ABB RAPID module: Module1.mod

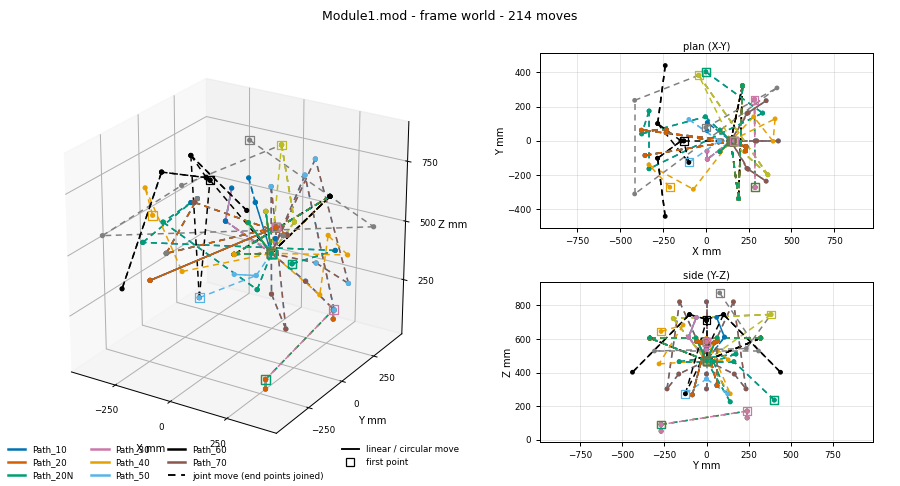
[picture p0: tool path of Module1.mod in frame world, 214 of 214 moves have a stored position in this frame; points joined in program order, loops and branches not executed]
MODULE Module1
    CONST robtarget p1:=[[392.068313627,0,352.752670777],[0,-0.707106781,0.707106781,0],[0,0,-1,0],[90,9E+09,9E+09,9E+09,9E+09,9E+09]];
    CONST robtarget p2:=[[0.889574022,-392.067304437,352.752670777],[0,-0.001134464,0.999999356,0],[-1,0,-1,0],[0.629463871,9E+09,9E+09,9E+09,9E+09,9E+09]];
    CONST robtarget p3:=[[218.23553446,-1.336915589,746.107847434],[0.698810372,0.082286187,0.062863115,0.707772051],[0,2,-1,4],[90.000000666,9E+09,9E+09,9E+09,9E+09,9E+09]];
    CONST robtarget Target_10:=[[521.001806146,0.000051805,471.113280829],[0.087155634,0.000000007,-0.996194708,0.000000054],[-2,1,0,4],[36.59813987,9E+09,9E+09,9E+09,9E+09,9E+09]];
    CONST robtarget Target_20:=[[285.146257362,-272.870516499,35.963966592],[0.000757376,0.999985094,-0.005407215,0.000030026],[-2,1,1,4],[5.849592085,9E+09,9E+09,9E+09,9E+09,9E+09]];
    CONST robtarget p_home:=[[146.001829286,-0.000011627,471.113261606],[0.087155743,-0.000000036,-0.996194698,0.000000029],[0,0,0,4],[89.999996076,9E+09,9E+09,9E+09,9E+09,9E+09]];
    CONST robtarget Target_30:=[[287.259986787,-269.999977839,91.999978977],[-0.000000081,1,-0.000000014,0.000000023],[1,-2,2,4],[-117.310008956,9E+09,9E+09,9E+09,9E+09,9E+09]];
    CONST robtarget p_1N:=[[8.64226597,106.715719366,611.703507902],[0.138141629,-0.665888474,0.721995202,0.127406274],[1,0,0,4],[175.197094616,9E+09,9E+09,9E+09,9E+09,9E+09]];
    CONST robtarget P_2N:=[[7.080305092,60.190965239,728.768322005],[0.731213881,0.142173983,-0.124037041,0.655536141],[1,2,-2,4],[175.262160505,9E+09,9E+09,9E+09,9E+09,9E+09]];
    CONST robtarget P_3N:=[[163.183896526,0.000014151,536.098477225],[0.0000012,0.727533257,0.000001374,0.686072416],[0,0,-2,5],[89.999982014,9E+09,9E+09,9E+09,9E+09,9E+09]];
    CONST robtarget p_1:=[[8.636290588,-106.716217244,611.703480594],[0.138137727,0.665909107,0.721976171,-0.127410507],[-1,0,0,4],[4.799479876,9E+09,9E+09,9E+09,9E+09,9E+09]];
    CONST robtarget p_2:=[[6.784511962,-60.211507569,728.777229645],[0.719966249,-0.13831615,-0.128050116,-0.667922459],[-1,-2,2,4],[4.731019989,9E+09,9E+09,9E+09,9E+09,9E+09]];
    CONST robtarget p_3:=[[163.183888274,0.000014151,536.098499129],[0.000000145,0.727533285,-0.000000052,0.686072386],[0,0,2,5],[89.99998012,9E+09,9E+09,9E+09,9E+09,9E+09]];
    CONST robtarget Target_40:=[[287.259965591,-270.000057213,52.000013466],[0.000000073,1,-0.000000039,-0.000000056],[1,-2,2,4],[-117.310020828,9E+09,9E+09,9E+09,9E+09,9E+09]];
    CONST robtarget Target_50:=[[284.216593063,241.497276454,171.455327595],[0.461769055,0.534075398,-0.465655163,0.533571062],[-1,2,2,4],[-62.533115785,9E+09,9E+09,9E+09,9E+09,9E+09]];
    CONST robtarget Target_60:=[[284.219997377,241.500021616,130.999992148],[0.46175743,0.534074104,-0.465673848,0.533566111],[-1,2,2,4],[-62.529982153,9E+09,9E+09,9E+09,9E+09,9E+09]];
    CONST robtarget V_1:=[[82.331083989,-62.999984967,606.511608487],[0.071559788,0.071559953,0.703476453,-0.703476545],[0,-1,0,4],[89.999987026,9E+09,9E+09,9E+09,9E+09,9E+09]];
    CONST robtarget V_1N:=[[82.331109479,63.000017394,606.51159395],[0.071560002,-0.071559898,0.703476541,0.703476442],[0,1,0,4],[89.999987026,9E+09,9E+09,9E+09,9E+09,9E+09]];
    CONST robtarget C_1:=[[191.190430031,-336.50536979,605.533784051],[0.764366784,0.298522446,0.400168922,-0.40803505],[-1,0,0,5],[43.240437571,9E+09,9E+09,9E+09,9E+09,9E+09]];
    CONST robtarget C_2:=[[214.025606426,322.463502613,605.533757072],[0.747963081,-0.184507274,0.463905018,0.437379047],[1,0,0,5],[136.981847176,9E+09,9E+09,9E+09,9E+09,9E+09]];
    CONST robtarget W_1:=[[247.316648717,-164.939578377,391.966969215],[0.113983949,0.287803778,0.950255151,-0.034522355],[0,0,0,4],[66.141884398,9E+09,9E+09,9E+09,9E+09,9E+09]];
    CONST robtarget W_2:=[[352.191610818,-234.882458107,303.624691389],[0.473921077,0.25183348,0.831490212,-0.143536542],[0,0,0,1],[80.737845767,9E+09,9E+09,9E+09,9E+09,9E+09]];
    CONST robtarget W_3:=[[239.99749851,-160.058376457,821.147940575],[0.957041414,-0.002116332,-0.006987781,-0.289859319],[0,0,0,1],[62.449758689,9E+09,9E+09,9E+09,9E+09,9E+09]];
    CONST robtarget W_1N:=[[247.316818335,164.939254461,391.966986138],[0.113983997,-0.287803395,0.950255264,0.034522268],[0,0,0,4],[113.858082982,9E+09,9E+09,9E+09,9E+09,9E+09]];
    CONST robtarget W_2N:=[[352.191752595,234.882274014,303.624688203],[0.473921109,-0.251833367,0.831490242,0.143536459],[0,0,0,1],[99.262132559,9E+09,9E+09,9E+09,9E+09,9E+09]];
    CONST robtarget W_3N:=[[239.997409078,160.058529004,821.147901462],[0.957041328,0.002116447,-0.006987768,0.289859602],[0,0,0,1],[117.550294272,9E+09,9E+09,9E+09,9E+09,9E+09]];
    CONST robtarget W_1M:=[[297.271872691,-0.000465817,391.966986138],[0.119097181,0.000000639,0.992882602,-0.000000091],[0,0,0,4],[89.999966529,9E+09,9E+09,9E+09,9E+09,9E+09]];
    CONST robtarget W_2M:=[[423.330501194,-0.000355239,303.624688203],[0.495180707,0.000000288,0.868790002,-0.000000146],[0,0,0,1],[89.999975658,9E+09,9E+09,9E+09,9E+09,9E+09]];
    CONST robtarget W_3M:=[[288.474416667,0.000127958,821.147901462],[0.999973346,0.000000058,-0.00730125,0.000000233],[0,0,0,1],[90.000034639,9E+09,9E+09,9E+09,9E+09,9E+09]];
    CONST robtarget X_1:=[[0,78.539559134,874.160589801],[0.691605325,-0.151532114,-0.151144716,-0.689837204],[-1,-2,2,4],[0,9E+09,9E+09,9E+09,9E+09,9E+09]];
    CONST robtarget X_2:=[[415.33755253,309.389185706,528.887172849],[0.849004005,-0.453249239,0.240111488,-0.126900749],[-1,-2,2,4],[40.681857579,9E+09,9E+09,9E+09,9E+09,9E+09]];
    CONST robtarget X_3:=[[-415.337536047,-309.389266315,528.887209232],[0.126900628,-0.240111463,-0.453249193,0.849004055],[1,-2,2,4],[-139.318142179,9E+09,9E+09,9E+09,9E+09,9E+09]];
    CONST robtarget X_4:=[[-415.337536047,236.913158737,543.685581945],[0.101780243,0.251789726,-0.356952968,-0.893771388],[1,-2,2,0],[-50.763285478,9E+09,9E+09,9E+09,9E+09,9E+09]];
    CONST robtarget X_5:=[[-41.445591379,383.178553538,745.950183931],[0.84767252,-0.258823437,-0.399440963,0.234325935],[1,0,2,2],[-98.481786712,9E+09,9E+09,9E+09,9E+09,9E+09]];
    CONST robtarget X_6:=[[362.018169952,-197.519749184,722.249115014],[0.304749808,-0.447145216,0.085266241,-0.836611247],[-1,0,0,3],[-38.266919692,9E+09,9E+09,9E+09,9E+09,9E+09]];
    CONST robtarget X_1N:=[[0.000000834,403.15639969,237.203949931],[0.073790046,0.703246065,-0.703246066,0.073790047],[1,2,-2,1],[179.999999425,9E+09,9E+09,9E+09,9E+09,9E+09]];
    CONST robtarget X_2N:=[[331.55662683,162.653720049,465.432471111],[0.252272501,-0.100646522,0.893893602,-0.356627385],[1,2,-2,1],[60.822047557,9E+09,9E+09,9E+09,9E+09,9E+09]];
    CONST robtarget X_3N:=[[-331.55662683,-162.653720049,465.432471111],[0.356627385,-0.893893602,-0.100646522,0.252272501],[-1,2,-2,1],[-119.177952443,9E+09,9E+09,9E+09,9E+09,9E+09]];
    CONST robtarget X_4N:=[[-331.250610789,174.805835636,510.726475074],[0.339834937,0.900284398,-0.08567432,-0.25818623],[-1,2,-2,5],[-63.659993257,9E+09,9E+09,9E+09,9E+09,9E+09]];
    CONST robtarget X_5N:=[[-374.440005394,41.091313566,465.564181588],[0.749183837,-0.161989044,-0.583991849,0.267276351],[1,0,-1,5],[-100.774260558,9E+09,9E+09,9E+09,9E+09,9E+09]];
    CONST robtarget X_6N:=[[-2.632659202,140.822678333,226.6540893],[0.40289172,-0.791073566,0.406435971,-0.216080255],[2,-1,1,4],[-134.924368397,9E+09,9E+09,9E+09,9E+09,9E+09]];
    CONST robtarget Y_1:=[[-210.120078432,-270.066474725,645.109260776],[0.645899113,-0.294294368,-0.689526235,0.14407891],[0,-1,-1,4],[38.496984805,9E+09,9E+09,9E+09,9E+09,9E+09]];
    CONST robtarget Y_2:=[[-332.251792218,-139.221948013,683.413400446],[0.397666016,-0.607257591,-0.672511001,0.144322248],[0,-1,-1,4],[32.37384699,9E+09,9E+09,9E+09,9E+09,9E+09]];
    CONST robtarget Y_3:=[[-72.630364019,-282.279817743,452.062943225],[0.811290854,0.182756719,-0.544569242,0.108864467],[0,-1,-1,4],[67.302510587,9E+09,9E+09,9E+09,9E+09,9E+09]];
    CONST robtarget Y_1N:=[[404.369104364,129.154096097,476.680005353],[0.53756367,0.17326855,0.59287786,-0.574020168],[0,-1,1,0],[134.749695485,9E+09,9E+09,9E+09,9E+09,9E+09]];
    CONST robtarget Y_2N:=[[392.48212923,-1.905303197,603.414236241],[0.46076172,0.535801826,0.564446059,-0.426632965],[0,-1,1,0],[145.341252401,9E+09,9E+09,9E+09,9E+09,9E+09]];
    CONST robtarget Y_3N:=[[279.346088031,141.147078038,274.585862253],[0.503356617,-0.339132534,0.489277349,-0.626281819],[0,-1,1,0],[94.902982809,9E+09,9E+09,9E+09,9E+09,9E+09]];
    CONST robtarget Z_2:=[[-99.128387414,-125.510607371,274.499713941],[0.416432493,-0.413921608,-0.760020488,-0.278606783],[0,0,0,4],[-7.372818271,9E+09,9E+09,9E+09,9E+09,9E+09]];
    CONST robtarget Z_1:=[[78.954041542,-0.000003827,362.438821557],[0.320396549,-0.000000064,-0.947283512,-0.000000026],[0,0,0,4],[89.999981837,9E+09,9E+09,9E+09,9E+09,9E+09]];
    CONST robtarget Z_3:=[[-99.137091685,125.515849566,274.498901113],[0.416446875,0.4139185,-0.760023579,0.278581471],[0,0,0,4],[-172.625930856,9E+09,9E+09,9E+09,9E+09,9E+09]];
    CONST robtarget ZX_1:=[[-128.511903406,0.000190761,711.083912245],[0.884487955,-0.000000053,0.466563026,-0.000000381],[0,0,0,4],[89.999985014,9E+09,9E+09,9E+09,9E+09,9E+09]];
    CONST robtarget ZX_2:=[[-144.51454504,0.000201847,717.643201062],[0.894349523,-0.000000058,0.447368897,-0.000000382],[0,0,0,4],[89.99998573,9E+09,9E+09,9E+09,9E+09,9E+09]];
    CONST robtarget ZX_3:=[[-281.51246386,-101.104994512,745.706716204],[0.524000006,0.209719662,0.262113725,-0.782775863],[0,-1,0,4],[89.999986181,9E+09,9E+09,9E+09,9E+09,9E+09]];
    CONST robtarget ZX_4:=[[-237.121272697,-440.256288518,402.662256079],[0.383663649,0.438416509,0.653350112,-0.483452996],[0,-1,0,4],[42.187315149,9E+09,9E+09,9E+09,9E+09,9E+09]];
    CONST robtarget ZX_5:=[[-281.050992666,101.259764874,745.61212211],[0.525685714,-0.209366234,0.262956978,0.781456293],[0,1,0,4],[89.999982012,9E+09,9E+09,9E+09,9E+09,9E+09]];
    CONST robtarget ZX_6:=[[-236.656037874,440.177228205,402.542254003],[0.385192656,-0.438951233,0.653316343,0.481794757],[0,1,0,4],[137.807682603,9E+09,9E+09,9E+09,9E+09,9E+09]];
    CONST robtarget p_home_3:=[[166.000125891,0.00020889,583.659974997],[0.085243027,0.000000334,-0.996360189,0.000000157],[0,0,0,4],[90.000018518,9E+09,9E+09,9E+09,9E+09,9E+09]];
    CONST robtarget Target_200:=[[-354.773050451,-84.344694535,268.460118696],[0.238303291,0.897110267,-0.306353089,0.211074619],[0,0,0,4],[-83.285519162,9E+09,9E+09,9E+09,9E+09,9E+09]];
    CONST robtarget Target_210:=[[-376.101703234,62.461413187,323.329887525],[0.610356235,0.09434494,-0.761034646,-0.198470569],[0,0,2,5],[-97.549460724,9E+09,9E+09,9E+09,9E+09,9E+09]];
    CONST robtarget Target_220:=[[-228.615156881,64.710223321,589.463784633],[0.883682757,-0.006763798,-0.415927533,-0.214623677],[0,0,2,1],[-96.203851173,9E+09,9E+09,9E+09,9E+09,9E+09]];
    CONST robtarget Target_230:=[[-231.243499004,47.678924526,579.148047545],[0.689418524,0.529628593,-0.314309158,-0.381320606],[0,3,2,1],[-96.314756715,9E+09,9E+09,9E+09,9E+09,9E+09]];
    CONST robtarget Target_240:=[[233.811720631,-32.846891162,579.148097614],[0.359150346,0.297266434,0.539378713,0.701223431],[-2,3,2,1],[89.465102118,9E+09,9E+09,9E+09,9E+09,9E+09]];
    CONST robtarget Target_400:=[[232.232129712,-57.590953584,586.336983128],[0.07210896,0.444347139,-0.20482834,0.869138233],[-2,0,2,1],[89.943689306,9E+09,9E+09,9E+09,9E+09,9E+09]];
    CONST robtarget Target_410:=[[232.232108838,-57.590933187,586.336951717],[0.41742242,-0.258654069,0.415327716,-0.765741134],[-2,0,-1,1],[89.943687469,9E+09,9E+09,9E+09,9E+09,9E+09]];
    CONST robtarget Target_420:=[[233.81605987,-32.995526687,579.458327437],[0.090145667,-0.543431647,-0.279179277,-0.786520651],[-2,3,-1,1],[89.893000259,9E+09,9E+09,9E+09,9E+09,9E+09]];

    PROC Path_10()
        MoveJ p_home,v800,fine,tool0\WObj:=wobj0;
        MoveJ p_1,v800,fine,tool0\WObj:=wobj0;
        MoveJ p_2,v7000,fine,tool0\WObj:=wobj0;
        MoveJ p_1,v7000,fine,tool0\WObj:=wobj0;
        MoveJ p_home,v3000,fine,tool0\WObj:=wobj0;
        MoveJ p_3,v1000,fine,tool0\WObj:=wobj0;
        MoveJ p_home,v40,fine,tool0\WObj:=wobj0;
        MoveJ p_1N,v800,fine,tool0\WObj:=wobj0;
        MoveJ P_2N,v7000,fine,tool0\WObj:=wobj0;
        MoveJ p_1N,v7000,fine,tool0\WObj:=wobj0;
        MoveJ p_home,v3000,fine,tool0\WObj:=wobj0;
        MoveJ P_3N,v1000,fine,tool0\WObj:=wobj0;
        MoveJ p_home,v40,fine,tool0\WObj:=wobj0;
    ENDPROC
    PROC Path_20()
        MoveJ Target_30,v1000,fine,Servo\WObj:=wobj0;
        MoveL Target_40,v1000,fine,Servo\WObj:=wobj0;
        g_GripIn;
        SetDO gripper,1;
        MoveL Target_30,v1000,fine,Servo\WObj:=wobj0;
        MoveJ Target_50,v1000,fine,Camera\WObj:=wobj0;
        MoveL Target_60,v1000,fine,Camera\WObj:=wobj0;
        g_GripOut;
        SetDO gripper,0;
        MoveL Target_50,v1000,fine,Camera\WObj:=wobj0;
    ENDPROC
    PROC Path_20N()
        MoveJ Target_30,v1000,fine,Servo\WObj:=wobj0;
        MoveL Target_40,v1000,fine,Servo\WObj:=wobj0;
        MoveL Target_30,v1000,fine,Servo\WObj:=wobj0;
        MoveJ Target_50,v1000,fine,Camera\WObj:=wobj0;
        MoveL Target_60,v1000,fine,Camera\WObj:=wobj0;
        MoveL Target_50,v1000,fine,Camera\WObj:=wobj0;
    ENDPROC
    PROC Path_30()
        MoveJ p_home,v800,fine,tool0\WObj:=wobj0;
        MoveJ p_1,v800,fine,tool0\WObj:=wobj0;
        MoveJ p_2,v7000,fine,tool0\WObj:=wobj0;
        MoveJ p_1,v7000,fine,tool0\WObj:=wobj0;
        MoveJ p_home,v3000,fine,tool0\WObj:=wobj0;
        MoveJ P_3N,v5,fine,tool0\WObj:=wobj0;
        MoveJ p_home,v5,fine,tool0\WObj:=wobj0;
    ENDPROC
    PROC Path_40()
        MoveL p_home,v1000,fine,Servo\WObj:=wobj0;
        MoveL V_1,v60,fine,Servo\WObj:=wobj0;
        MoveL p_home,v60,fine,Servo\WObj:=wobj0;
        MoveL V_1N,v60,fine,Servo\WObj:=wobj0;
        MoveJ p_home,v60,fine,Servo\WObj:=wobj0;
        MoveJ C_1,v1000,fine,Servo\WObj:=wobj0;
        MoveJ C_2,v1000,fine,Servo\WObj:=wobj0;
        MoveJ p_home,v1000,fine,Servo\WObj:=wobj0;
        MoveJ C_2,v1000,fine,Servo\WObj:=wobj0;
        MoveJ C_1,v1000,fine,Servo\WObj:=wobj0;
        MoveJ p_home,v1000,fine,Servo\WObj:=wobj0;
        MoveJ C_2,v1000,fine,Servo\WObj:=wobj0;
        MoveJ C_1,v1000,fine,Servo\WObj:=wobj0;
        MoveJ p_home,v1000,fine,Servo\WObj:=wobj0;
        MoveJ C_1,v1000,fine,Servo\WObj:=wobj0;
        MoveJ C_2,v1000,fine,Servo\WObj:=wobj0;
        MoveJ p_home,v1000,fine,Servo\WObj:=wobj0;
    ENDPROC
    PROC Path_50()
        MoveJ p_home,v1000,fine,Servo\WObj:=wobj0;
        MoveJ W_1,v1000,fine,Servo\WObj:=wobj0;
        MoveJ W_2,v1000,fine,Servo\WObj:=wobj0;
        MoveJ W_3,v1000,fine,Servo\WObj:=wobj0;
        MoveJ p_home,v1000,fine,Servo\WObj:=wobj0;
        MoveJ W_1N,v1000,fine,Servo\WObj:=wobj0;
        MoveJ W_2N,v1000,fine,Servo\WObj:=wobj0;
        MoveJ W_3N,v1000,fine,Servo\WObj:=wobj0;
        MoveJ p_home,v1000,fine,Servo\WObj:=wobj0;
        MoveJ W_1M,v1000,fine,Servo\WObj:=wobj0;
        MoveJ W_2M,v1000,fine,Servo\WObj:=wobj0;
        MoveJ W_3M,v1000,fine,Servo\WObj:=wobj0;
        MoveJ p_home,v1000,fine,Servo\WObj:=wobj0;
        MoveJ W_1M,v1000,fine,Servo\WObj:=wobj0;
        MoveJ W_2M,v1000,fine,Servo\WObj:=wobj0;
        MoveJ W_3M,v1000,fine,Servo\WObj:=wobj0;
        MoveJ p_home,v500,fine,Servo\WObj:=wobj0;
    ENDPROC
    PROC Path_60()
        MoveJ p_home,v1000,fine,Servo\WObj:=wobj0;
        MoveJ C_1,v1000,fine,Servo\WObj:=wobj0;
        MoveJ C_2,v1000,fine,Servo\WObj:=wobj0;
        MoveJ p_home,v1000,fine,Servo\WObj:=wobj0;
        MoveJ C_2,v1000,fine,Servo\WObj:=wobj0;
        MoveJ C_1,v1000,fine,Servo\WObj:=wobj0;
        MoveJ p_home,v1000,fine,Servo\WObj:=wobj0;
        MoveJ C_2,v1000,fine,Servo\WObj:=wobj0;
        MoveJ C_1,v1000,fine,Servo\WObj:=wobj0;
        MoveJ p_home,v1000,fine,Servo\WObj:=wobj0;
        MoveJ C_1,v1000,fine,Servo\WObj:=wobj0;
        MoveJ C_2,v1000,fine,Servo\WObj:=wobj0;
        MoveJ p_home,v1000,fine,Servo\WObj:=wobj0;
    ENDPROC
    PROC Path_70()
        MoveJ p_home,v1000,fine,Servo\WObj:=wobj0;
        MoveJ W_1,v1000,fine,Servo\WObj:=wobj0;
        MoveJ W_2,v1000,fine,Servo\WObj:=wobj0;
        MoveJ W_3,v1000,fine,Servo\WObj:=wobj0;
        MoveJ p_home,v1000,fine,Servo\WObj:=wobj0;
        MoveJ W_1N,v1000,fine,Servo\WObj:=wobj0;
        MoveJ W_2N,v1000,fine,Servo\WObj:=wobj0;
        MoveJ W_3N,v1000,fine,Servo\WObj:=wobj0;
        MoveJ p_home,v1500,fine,Servo\WObj:=wobj0;
        MoveJ W_1M,v1500,fine,Servo\WObj:=wobj0;
        MoveJ W_2M,v1500,fine,Servo\WObj:=wobj0;
        MoveJ W_3M,v1500,fine,Servo\WObj:=wobj0;
        MoveJ p_home,v1500,fine,Servo\WObj:=wobj0;
    ENDPROC
    PROC Path_80()
        MoveJ X_1,v2500,z100,Servo\WObj:=wobj0;
        MoveJ X_2,v2500,z100,Servo\WObj:=wobj0;
        MoveJ X_3,v2500,z100,Servo\WObj:=wobj0;
        MoveJ X_4,v2500,z100,Servo\WObj:=wobj0;
        MoveJ X_5,v2500,z100,Servo\WObj:=wobj0;
        MoveJ X_6,v2500,z100,Servo\WObj:=wobj0;
        MoveJ p_home,v2500,z100,Servo\WObj:=wobj0;
    ENDPROC
    PROC Path_90()
        MoveJ X_5,v2500,z100,Servo\WObj:=wobj0;
        MoveJ X_6,v2500,z100,Servo\WObj:=wobj0;
        MoveJ p_home,v2500,z100,Servo\WObj:=wobj0;
        MoveJ X_5,v2500,z100,Servo\WObj:=wobj0;
        MoveJ X_6,v2500,z100,Servo\WObj:=wobj0;
        MoveJ p_home,v2500,z100,Servo\WObj:=wobj0;
    ENDPROC
    PROC Path_100()
        MoveJ X_1N,v2500,z100,Servo\WObj:=wobj0;
        MoveJ X_2N,v2500,z100,Servo\WObj:=wobj0;
        MoveJ X_3N,v2500,z100,Servo\WObj:=wobj0;
        MoveJ X_4N,v2500,z100,Servo\WObj:=wobj0;
        MoveJ X_5N,v2500,z100,Servo\WObj:=wobj0;
        MoveJ X_6N,v2500,z100,Servo\WObj:=wobj0;
        MoveJ p_home,v2500,z100,Servo\WObj:=wobj0;
    ENDPROC
    PROC Path_110()
        MoveL p_home,v1000,fine,Servo\WObj:=wobj0;
        MoveL V_1,v60,fine,Servo\WObj:=wobj0;
        MoveL p_home,v60,fine,Servo\WObj:=wobj0;
        MoveL V_1N,v60,fine,Servo\WObj:=wobj0;
        MoveJ p_home,v60,fine,Servo\WObj:=wobj0;
        MoveJ C_1,v1000,fine,Servo\WObj:=wobj0;
        MoveJ C_2,v1000,fine,Servo\WObj:=wobj0;
    ENDPROC
     PROC Path_120()
        MoveJ X_1N,v2500,z100,Servo\WObj:=wobj0;
        MoveJ X_2N,v2500,z100,Servo\WObj:=wobj0;
        MoveJ X_3N,v2500,z100,Servo\WObj:=wobj0;
        MoveJ X_4N,v2500,z100,Servo\WObj:=wobj0;
        MoveJ X_5N,v2500,z100,Servo\WObj:=wobj0;
        MoveJ X_6N,v2500,z100,Servo\WObj:=wobj0;
        MoveJ p_home,v1500,z100,Servo\WObj:=wobj0;
    ENDPROC
    PROC Path_20B()
        MoveJ Target_50,v1000,fine,Servo\WObj:=wobj0;
        MoveL Target_60,v1000,fine,Servo\WObj:=wobj0;
        MoveL Target_50,v1000,fine,Servo\WObj:=wobj0;
        MoveJ Target_30,v1000,fine,Servo\WObj:=wobj0;
        MoveL Target_40,v1000,fine,Servo\WObj:=wobj0;
        MoveL Target_30,v1000,fine,Servo\WObj:=wobj0;
    ENDPROC
    PROC Path_130()
        MoveJ Y_1,v1000,z100,Servo\WObj:=wobj0;
        MoveJ Y_2,v1000,z100,Servo\WObj:=wobj0;
        MoveJ Y_3,v500,z100,Servo\WObj:=wobj0;
        MoveJ p_home,v1000,z100,Servo\WObj:=wobj0;
        MoveJ Y_1N,v1000,z100,Servo\WObj:=wobj0;
        MoveJ Y_2N,v1000,z100,Servo\WObj:=wobj0;
        MoveJ Y_3N,v500,z100,Servo\WObj:=wobj0;
        MoveJ p_home,v1000,z100,Servo\WObj:=wobj0;
    ENDPROC
    PROC Path_140()
        MoveJ Z_2,v500,fine,Servo\WObj:=wobj0;
        MoveJ Z_1,v500,fine,Servo\WObj:=wobj0;
        MoveJ Z_3,v500,fine,Servo\WObj:=wobj0;
        MoveJ Z_1,v500,fine,Servo\WObj:=wobj0;
        MoveJ p_home,v500,fine,Servo\WObj:=wobj0;
    ENDPROC
    PROC Path_150()
        MoveJ ZX_1,v1000,z100,Servo\WObj:=wobj0;
        MoveJ ZX_2,v1000,z100,Servo\WObj:=wobj0;
        MoveJ ZX_3,v1000,z100,Servo\WObj:=wobj0;
        MoveJ ZX_4,v1000,z100,Servo\WObj:=wobj0;
        MoveJ ZX_3,v1000,z100,Servo\WObj:=wobj0;
        MoveJ ZX_2,v1000,z100,Servo\WObj:=wobj0;
        MoveJ ZX_5,v1000,z100,Servo\WObj:=wobj0;
        MoveJ ZX_6,v1000,z100,Servo\WObj:=wobj0;
        MoveJ ZX_5,v1000,z100,Servo\WObj:=wobj0;
        MoveJ Z_2,v1000,z100,Servo\WObj:=wobj0;
        MoveJ ZX_1,v1000,z100,Servo\WObj:=wobj0;
        MoveJ p_home,v1000,z100,Servo\WObj:=wobj0;
    ENDPROC
    PROC Path_556()
        MoveJ p_home_3,v1000,z100,tool0\WObj:=wobj0;
        MoveJ Target_200,v7000,z100,tool0\WObj:=wobj0;
        MoveJ p_home_3,v7000,z100,tool0\WObj:=wobj0;
        MoveJ Target_210,v7000,z100,tool0\WObj:=wobj0;
        MoveJ Target_220,v1000,z100,tool0\WObj:=wobj0;
        MoveJ Target_230,v1000,z100,tool0\WObj:=wobj0;
        MoveJ Target_240,v1000,z100,tool0\WObj:=wobj0;
        MoveJ Target_400,v1000,z100,tool0\WObj:=wobj0;
        MoveJ Target_410,v1000,z100,tool0\WObj:=wobj0;
        MoveJ Target_420,v1000,z100,tool0\WObj:=wobj0;
    ENDPROC
    PROC Path_557()
        MoveJ p_home_3,v1000,z100,tool0\WObj:=wobj0;
        MoveJ Target_200,v7000,z100,tool0\WObj:=wobj0;
        MoveJ p_home_3,v7000,z100,tool0\WObj:=wobj0;
        MoveJ Target_210,v7000,z100,tool0\WObj:=wobj0;
        MoveJ Target_220,v1000,z100,tool0\WObj:=wobj0;
        MoveJ Target_230,v1000,z100,tool0\WObj:=wobj0;
        MoveJ Target_240,v1000,z100,tool0\WObj:=wobj0;
        MoveJ Target_400,v1000,z100,tool0\WObj:=wobj0;
        MoveJ Target_410,v1000,z100,tool0\WObj:=wobj0;
        MoveJ Target_420,v1000,z100,tool0\WObj:=wobj0;
        MoveJ p_home_3,v1000,z100,tool0\WObj:=wobj0;
    ENDPROC
     PROC Path_558()
        MoveL p_home,v3000,fine,Servo\WObj:=wobj0;
        MoveL V_1,v3000,fine,Servo\WObj:=wobj0;
        MoveL p_home,v3000,fine,Servo\WObj:=wobj0;
        MoveL V_1N,v3000,fine,Servo\WObj:=wobj0;
        MoveJ p_home,v3000,fine,Servo\WObj:=wobj0;
        MoveJ C_1,v3000,fine,Servo\WObj:=wobj0;
        MoveJ C_2,v3000,fine,Servo\WObj:=wobj0;
    ENDPROC
    PROC Path_566()
        MoveJ p_home_3,v2000,z100,tool0\WObj:=wobj0;
        MoveJ Target_200,v7000,z100,tool0\WObj:=wobj0;
        MoveJ p_home_3,v7000,z100,tool0\WObj:=wobj0;
        MoveJ Target_210,v7000,z100,tool0\WObj:=wobj0;
        MoveJ Target_220,v2000,z100,tool0\WObj:=wobj0;
        MoveJ Target_230,v2000,z100,tool0\WObj:=wobj0;
        MoveJ Target_240,v2000,z100,tool0\WObj:=wobj0;
        MoveJ Target_400,v2000,z100,tool0\WObj:=wobj0;
        MoveJ Target_410,v2000,z100,tool0\WObj:=wobj0;
        MoveJ Target_420,v2000,z100,tool0\WObj:=wobj0;
    ENDPROC
    PROC Path_567()
        MoveJ p_home_3,v2000,z100,tool0\WObj:=wobj0;
        MoveJ Target_200,v2000,z100,tool0\WObj:=wobj0;
        MoveJ p_home_3,v2000,z100,tool0\WObj:=wobj0;
        MoveJ Target_210,v2000,z100,tool0\WObj:=wobj0;
        MoveJ Target_220,v2000,z100,tool0\WObj:=wobj0;
        MoveJ Target_230,v2000,z100,tool0\WObj:=wobj0;
        MoveJ Target_240,v2000,z100,tool0\WObj:=wobj0;
        MoveJ Target_400,v2000,z100,tool0\WObj:=wobj0;
        MoveJ Target_410,v2000,z100,tool0\WObj:=wobj0;
        MoveJ Target_420,v2000,z100,tool0\WObj:=wobj0;
        MoveJ p_home_3,v2000,z100,tool0\WObj:=wobj0;
    ENDPROC
     PROC Path_568()
        MoveL p_home,v5000,fine,Servo\WObj:=wobj0;
        MoveL V_1,v5000,fine,Servo\WObj:=wobj0;
        MoveL p_home,v5000,fine,Servo\WObj:=wobj0;
        MoveL V_1N,v5000,fine,Servo\WObj:=wobj0;
        MoveJ p_home,v5000,fine,Servo\WObj:=wobj0;
        MoveJ C_1,v5000,fine,Servo\WObj:=wobj0;
        MoveJ C_2,v5000,fine,Servo\WObj:=wobj0;
    ENDPROC
    PROC Path_Home()
        MoveJ p_home_3,v2000,z100,tool0\WObj:=wobj0;
    ENDPROC
ENDMODULE
